// TwinCAT 3 PLC project Tc3_Sqlite
// Title: Tc3_Sqlite
// Company: Chua Siang Poh
// ProjectVersion: 1.0
// ProgramVersion: 3.1.0.8
// libraries:
//   Tc2_Database, * (Beckhoff Automation GmbH)
//   Tc2_Standard, * (Beckhoff Automation GmbH)
//   Tc2_System, * (Beckhoff Automation GmbH)
//   Tc3_Interfaces, * (Beckhoff Automation GmbH)
//   Tc3_Module, * (Beckhoff Automation GmbH)
// project tree:
//   Custom Datatypes/ DB_FunctionResult.TcDUT (not stored)
//   / DBAdaptor.TcPOU, MAIN.TcPOU, PlcTask.TcTTO
//   Interfaces/ ITF_DBAdaptor.TcIO (not stored)
//   Version/ Global_Version.TcGVL
// real-time tasks:
//   TASK PlcTask: cycle T#10ms, priority 20, ADS port 350

CONFIGURATION Tc3_Sqlite
    RESOURCE PLC ON TwinCAT3
        TASK PlcTask(INTERVAL := T#10ms, PRIORITY := 20);
        PROGRAM MAIN WITH PlcTask : MAIN;
    END_RESOURCE
END_CONFIGURATION

// ---- Version/Global_Version.TcGVL
// This function has been automatically generated from the project information.
VAR_GLOBAL CONSTANT
	{attribute 'const_non_replaced'}
	stLibVersion_Tc3_Sqlite : ST_LibVersion := (iMajor := 1, iMinor := 0, iBuild := 0, iRevision := 0, sVersion := '1.0');
END_VAR

// ---- MAIN.TcPOU
PROGRAM MAIN
VAR
	myDB	: DBAdaptor;
	fbTon 	: TON;
	fbTrig	: R_TRIG;
	SQL : STRING(255) := 'INSERT INTO messagelog (message,timestamp) VALUES($'Interval Triggered$',datetime($'now$'))';
	Debug : DB_FunctionResult;
END_VAR

ACT_Interval();
myDB.udiDatabase_ID := 1;
myDB.TimeOut := T#5S;
IF fbTrig.Q THEN
	Debug := myDB.SQL_Insert(SQL);
END_IF

ACTION ACT_Interval:
fbTon(IN:= NOT fbTon.Q, PT:= T#1S );
fbTrig(CLK:= fbTon.Q);
END_ACTION

END_PROGRAM

// ---- DBAdaptor.TcPOU
//{attribute 'hide_all_locals'}
FUNCTION_BLOCK PUBLIC DBAdaptor IMPLEMENTS ITF_DBAdaptor
VAR_INPUT
END_VAR
VAR_OUTPUT
END_VAR
VAR
	Database_Id	: UDINT := 0;
	sAmsNetId	: STRING(23) := '';
	tTimeOut	: TIME := T#1S;
	fbOpenConn	: FB_DBConnectionOpen;
	fbCloseConn	: FB_DBConnectionClose;
	fbAddConn	: FB_DBConnectionAdd;
	fbSqlDelete : FB_DBRecordDelete;
	fbSqlInsert : FB_DBRecordInsert_EX;
	fbSqlSelect : FB_DBRecordArraySelect;
	iState 		: INT := 0;
END_VAR

;

{attribute 'object_name' := 'Close'}
METHOD PRIVATE Close : DB_FunctionResult
VAR_INPUT
END_VAR
fbCloseConn(
	sNetID:= sAmsNetID, 
	hDBID:= Database_ID, 
	bExecute:= TRUE, 
	tTimeout:= tTimeOut );
IF fbCloseConn.bBusy OR fbCloseConn.bError THEN 
	IF fbCloseConn.bError THEN 
		Close := DB_FunctionResult.DB_Error;
		fbCloseConn(
			sNetID:= sAmsNetId, 
			hDBID:= Database_ID, 
			bExecute:= FALSE, 
			tTimeout:= tTimeOut );
	END_IF
	IF fbCloseConn.bBusy THEN 
		Close := DB_FunctionResult.DB_Busy;
	END_IF
ELSE
	fbCloseConn(
		sNetID:= sAmsNetId, 
		hDBID:= Database_ID, 
		bExecute:= FALSE, 
		tTimeout:= tTimeOut );
	Close := DB_FunctionResult.DB_Ok;
END_IF
END_METHOD

{attribute 'object_name' := 'SQL_Delete'}
METHOD SQL_Delete : DB_FunctionResult
VAR_INPUT
	SQL : STRING(255);
END_VAR
END_METHOD

PROPERTY sNetID : STRING(23)
SET
sAmsNetId := sNetID;
END_SET
GET
sNetId := sAmsNetID;
END_GET
END_PROPERTY

{attribute 'object_name' := 'SQL_Insert'}
METHOD SQL_Insert : DB_FunctionResult
VAR_INPUT
	SQL : STRING(255);
END_VAR
fbSqlInsert(
	sNetID:= sAmsNetId, 
	hDBID:= Database_Id, 
	pCmdAddr:= ADR(SQL), 
	cbCmdSize:= SIZEOF(SQL), 
	bExecute:= TRUE, 
	tTimeout:= tTimeOut );
IF fbSqlInsert.bBusy OR fbSqlInsert.bError THEN
	IF fbSqlInsert.bError THEN
		fbSqlInsert(
			sNetID:= sAmsNetId, 
			hDBID:= Database_Id, 
			pCmdAddr:= ADR(SQL), 
			cbCmdSize:= SIZEOF(SQL), 
			bExecute:= FALSE, 
			tTimeout:= tTimeOut );
		SQL_Insert := DB_FunctionResult.DB_Error;
	END_IF
	IF fbSqlInsert.bBusy THEN
		SQL_Insert := DB_FunctionResult.DB_Busy;
	END_IF
ELSE
	fbSqlInsert(
		sNetID:= sAmsNetId, 
		hDBID:= Database_Id, 
		pCmdAddr:= ADR(SQL), 
		cbCmdSize:= SIZEOF(SQL), 
		bExecute:= FALSE, 
		tTimeout:= tTimeOut );
	SQL_Insert := DB_FunctionResult.DB_Ok;
END_IF
END_METHOD

{attribute 'object_name' := 'SQL_Select'}
METHOD SQL_Select : DB_FunctionResult
VAR_INPUT
	SQL 				: STRING(255);
	START_INDEX			: UDINT;
	ROWS				: UDINT;
	ROW_DATA_BYTES		: UDINT;
	ptr_ReceiveBuffer	: POINTER TO BYTE;
END_VAR
fbSqlSelect(
	sNetID:= sAmsNetId, 
	hDBID:= Database_ID, 
	pCmdAddr:= ADR(SQL), 
	cbCmdSize:= SIZEOF(SQL), 
	nStartIndex:= START_INDEX, 
	nRecordCount:= ROWS, 
	pDestAddr:= ptr_ReceiveBuffer, 
	cbRecordArraySize:= ROW_DATA_BYTES, 
	bExecute:= TRUE, 
	tTimeout:= tTimeOut );
IF fbSqlSelect.bBusy OR fbSqlSelect.bError THEN
	IF fbSqlSelect.bError THEN
		fbSqlSelect(
			sNetID:= sAmsNetId, 
			hDBID:= Database_ID, 
			pCmdAddr:= ADR(SQL), 
			cbCmdSize:= SIZEOF(SQL), 
			nStartIndex:= START_INDEX, 
			nRecordCount:= ROWS, 
			pDestAddr:= ptr_ReceiveBuffer, 
			cbRecordArraySize:= ROW_DATA_BYTES, 
			bExecute:= TRUE, 
			tTimeout:= tTimeOut );
		SQL_Select := DB_FunctionResult.DB_Error;
	END_IF
	IF fbSqlSelect.bBusy THEN
		SQL_Select := DB_FunctionResult.DB_Busy;
	END_IF
ELSE
	fbSqlSelect(
		sNetID:= sAmsNetId, 
		hDBID:= Database_ID, 
		pCmdAddr:= ADR(SQL), 
		cbCmdSize:= SIZEOF(SQL), 
		nStartIndex:= START_INDEX, 
		nRecordCount:= ROWS, 
		pDestAddr:= ptr_ReceiveBuffer, 
		cbRecordArraySize:= ROW_DATA_BYTES, 
		bExecute:= TRUE, 
		tTimeout:= tTimeOut );
	SQL_Select := DB_FunctionResult.DB_Ok;
END_IF
END_METHOD

{attribute 'object_name' := 'Open'}
METHOD PRIVATE Open : DB_FunctionResult
VAR_INPUT
END_VAR
fbOpenConn(
	sNetID:= sAmsNetId, 
	hDBID:= Database_ID, 
	bExecute:= TRUE, 
	tTimeout:= tTimeOut );
IF fbOpenConn.bBusy OR fbOpenConn.bError THEN 
	IF fbOpenConn.bError THEN 
		Open := DB_FunctionResult.DB_Error;
		fbOpenConn(
			sNetID:= sAmsNetId, 
			hDBID:= Database_ID, 
			bExecute:= FALSE, 
			tTimeout:= tTimeOut );
	END_IF
	IF fbOpenConn.bBusy THEN 
		Open := DB_FunctionResult.DB_Busy;
	END_IF
	
ELSE
	fbOpenConn(
		sNetID:= sAmsNetId, 
		hDBID:= Database_ID, 
		bExecute:= FALSE, 
		tTimeout:= tTimeOut );
	Open := DB_FunctionResult.DB_Ok;
END_IF
END_METHOD

PROPERTY udiDatabase_ID : UDINT
SET
Database_ID := udiDatabase_Id;
END_SET
GET
udiDatabase_ID := Database_Id;
END_GET
END_PROPERTY

PROPERTY TimeOut : TIME
GET
TimeOut := tTimeOut;
END_GET
SET
tTimeOut := TimeOut;
END_SET
END_PROPERTY

END_FUNCTION_BLOCK
